// TwinCAT 3 PLC project Untitled2
// ProgramVersion: 3.1.4023.0
// libraries:
//   Tc2_Standard, * (Beckhoff Automation GmbH)
//   Tc2_System, * (Beckhoff Automation GmbH)
//   Tc3_Module, * (Beckhoff Automation GmbH)
// project tree:
//   DUTs/ SensorBrands.TcDUT
//   / PlcTask.TcTTO
//   Segment1/ MAIN.TcPOU, POU.TcPOU, tASK1.TcPOU, task3.TcPOU, task4.TcPOU, task5.TcPOU
//   Segment2/ deg_to_rad.TcPOU, ST_Timer.TcDUT, task21.TcPOU, task22.TcPOU
//   Segment3/ caseTest.TcPOU, EmotorStatus.TcDUT, SmotorParameter.TcDUT, task31.TcPOU, updPar.TcPOU, updPar_1.TcPOU
// real-time tasks:
//   TASK PlcTask: cycle T#10ms, priority 20, ADS port 350
//   TASK PlcTask1: cycle T#10ms, priority 21, ADS port 351

CONFIGURATION Untitled2
    RESOURCE PLC ON TwinCAT3
        TASK PlcTask(INTERVAL := T#10ms, PRIORITY := 21);
        PROGRAM MAIN WITH PlcTask : MAIN;
    END_RESOURCE
END_CONFIGURATION

// ---- DUTs/SensorBrands.TcDUT
{attribute 'qualified_only'}
{attribute 'strict'}
TYPE SensorBrands :
(
	Sick,
	Pliz,
	Parker,
	Bosch
);
END_TYPE

// ---- Segment2/ST_Timer.TcDUT
TYPE ST_Timer :
STRUCT
	myTime : TIME := T#10S;
	fbTimeOn : TON := (PT := myTime);
	myBool : BOOL := TRUE;
END_STRUCT
END_TYPE

// ---- Segment3/EmotorStatus.TcDUT
{attribute 'qualified_only'}
{attribute 'strict'}
TYPE EmotorStatus :
(
	start := 0,
	running := 1,
	stopped := 2
);
END_TYPE

// ---- Segment3/SmotorParameter.TcDUT
TYPE SmotorParameter :
STRUCT
	max_speed : REAL := 100;
	min_speed : REAL := 1;
END_STRUCT
END_TYPE

// ---- Segment1/MAIN.TcPOU
PROGRAM MAIN
VAR
END_VAR

task31();
caseTest();

END_PROGRAM

// ---- Segment3/task31.TcPOU
PROGRAM task31
VAR
	stMotorPar : SmotorParameter;
	stMotorPar2 : SmotorParameter;
	fbRTrig : R_TRIG;
	myBool : BOOL := TRUE;
	newVal : REAL := 50;
	motSpeed : REAL;
	trigSig : BOOL;
END_VAR

fbRTrig(CLK := myBool, Q => trigSig);

updPar(bUpdateValue := trigSig, fNewVal := newVal, stMotorParameters := stMotorPar);
updPar_1(bUpdateValue := trigSig, fNewVal := newVal, stMotorParameters := stMotorPar2);

stMotorPar.max_speed;
stMotorPar2.max_speed;

END_PROGRAM

// ---- Segment3/updPar.TcPOU
FUNCTION updPar : REAL
VAR_INPUT
	bUpdateValue : BOOL;
	fNewVal : REAL;
	stMotorParameters : SmotorParameter;
END_VAR
VAR
END_VAR
VAR_OUTPUT
	curMotorSpeed : REAL;
END_VAR

IF (bUpdateValue = TRUE) THEN
	stMotorParameters.max_speed := fNewVal;
END_IF

END_FUNCTION

// ---- Segment3/updPar_1.TcPOU
FUNCTION updPar_1 : REAL
VAR_INPUT
	bUpdateValue : BOOL;
	fNewVal : REAL;
	stMotorParameters : REFERENCE TO SmotorParameter;
END_VAR
VAR
END_VAR
VAR_OUTPUT
	curMotorSpeed : REAL;
END_VAR

IF (bUpdateValue = TRUE) THEN
	stMotorParameters.max_speed := fNewVal;
END_IF

END_FUNCTION

// ---- Segment3/caseTest.TcPOU
PROGRAM caseTest
VAR
	motorStatus : EmotorStatus;
	shiftVal : INT := 0;
END_VAR

CASE shiftVal OF
	0: motorStatus := EmotorStatus.stopped;
	1: motorStatus := EmotorStatus.start;
	2: motorStatus := EmotorStatus.running;
END_CASE

END_PROGRAM

// ---- Segment1/POU.TcPOU
PROGRAM POU
VAR
	tVar : TIME := T#5S;
	nRefVar : REFERENCE TO TIME REF= tVar;
END_VAR

nRefVar := T#1S;

END_PROGRAM

// ---- Segment1/tASK1.TcPOU
PROGRAM tASK1
VAR
	dtVar : DATE_AND_TIME := DT#2023-02-07-13:10:00;
	pDateTime : POINTER TO DATE_AND_TIME;
END_VAR

pDateTime := ADR(dtVar);
pDateTime^ := DT#2023-02-09-15:31:19;

END_PROGRAM

// ---- Segment1/task3.TcPOU
PROGRAM task3
VAR
	dateArray : ARRAY[1..4] OF DATE := [D#2023-02-07, D#2023-02-08, D#2023-02-09, D#2023-02-10];
END_VAR

dateArray[3] := D#2023-02-25;

END_PROGRAM

// ---- Segment1/task4.TcPOU
PROGRAM task4
VAR
	sensor1 : SensorBrands;
END_VAR

sensor1 := SensorBrands.Parker;

END_PROGRAM

// ---- Segment1/task5.TcPOU
PROGRAM task5
VAR
	myTime : TIME := T#10S;
	fbTimeOn : TON := (PT := myTime);
	myBool : BOOL := TRUE;
END_VAR

fbTimeOn(IN := myBool);

END_PROGRAM

// ---- Segment2/deg_to_rad.TcPOU
FUNCTION deg_to_rad : REAL
VAR_INPUT
	motor_deg : REAL;
END_VAR
VAR
	deg_var : REAL := 180;
	rad_var : REAL := PI;
	conv_var : REAL := rad_var/deg_var;
END_VAR
VAR_OUTPUT
	motor_rad : REAL;
END_VAR

motor_rad := motor_deg * conv_var;

END_FUNCTION

// ---- Segment2/task21.TcPOU
PROGRAM task21
VAR
	stTimer2 : ST_Timer := (myTime := T#5S);
	fbTimeOff : TOF := (PT := stTimer2.myTime);
END_VAR

fbTimeOff(IN := stTimer2.myBool);

END_PROGRAM

// ---- Segment2/task22.TcPOU
PROGRAM task22
VAR
	myMotAng : REAL := 180;
	myMotAngNew : REAL; 
END_VAR

deg_to_rad(motor_deg := myMotAng, motor_rad => myMotAngNew);

END_PROGRAM
